TYPE E_SYSTEM_HandScannerBaudrate :
(
	E_HandScannerBaudrate_IDLE,
	E_HandScannerBaudrate_READ,
	E_HandScannerBaudrate_WRITE,
	E_HandScannerBaudrate_ERROR_READ,
	E_HandScannerBaudrate_ERROR_WRITE,
	E_HandScannerBaudrate_DONE
);
END_TYPE

(* stored: Version 1.1.0.1, ProductVersion 3.1.4024.15
   DUT E_SYSTEM_HandScannerBaudrate: Id {fe8ac897-06a0-4e93-9b77-0c6499999c36} *)
